FUNCTION_BLOCK Test_TStreamAdd_Read_LINT_CheckAlignment EXTENDS T_UnitTestBase
VAR
    Stream  : T_Stream(StreamLength := 2);
    ArgType : E_ArgTypeId := E_ArgTypeId.Type_LINT;
END_VAR

METHOD  Init
VAR_INPUT
END_VAR
END_METHOD

{attribute 'analysis' := '-33'} // inhibit unused variable warning
METHOD RunTest
Stream.Init(2);

Stream.Add_BYTE(123);// add a byte to test alignment checks...
Stream.Add_LINT(123456789);

Stream.SetReadPosition(0);

Stream.Read_BYTE();

// check next value...	
AssertEquals_LINT(Expected     := 123456789,
                            Actual       := Stream.Read_LINT(),
                            Message := 'Stream.Read_LINT()');

// check we are at the end of the stream..							
AssertEquals_UDINT(Expected     := Stream.StreamLength,
                             Actual       := Stream.ReadPosition,
                             Message := 'Stream.ReadPosition');

TestCompleted := TRUE;
END_METHOD

END_FUNCTION_BLOCK

(* stored: Version 1.1.0.1, ProductVersion 3.1.4024.12
   POU Test_TStreamAdd_Read_LINT_CheckAlignment: Id {d6d6802f-baa7-4bec-853f-403ea7ba6b41}, SpecialFunc None
   Method Init: Id {a636beb3-f7e6-4358-8db3-340237f210dd}
   Method RunTest: Id {aaef7578-8755-446b-a2e0-42f9fac505a4} *)
